// TIA Portal V20 export
TYPE "typeEstopFunction"
// Safety status of estop button
// stored: Access Published, IsFailsafeCompliant true, Namespace Safety
   STRUCT
      STO : Bool;   // STO, safet torque of for drives
      released { ExternalWritable := 'False'} : Bool;   // Button OK
      ackReq { ExternalWritable := 'False'} : Bool;   // Acknowledge required
   END_STRUCT;
END_TYPE
